Staubli VAL3: onExit.pgx

program onExit()
begin
  // save it
  saveData:libSave()
  use:bUseRefresh=true
end
